// TIA Portal V16 program export: 1 tag tables, 0 data types, 0 data blocks, 2 code blocks (in call order from the OBs), 11 instance data blocks

VAR_GLOBAL   // PLC tag table "Standard-Variablentabelle"
   start AT %I0.4 : Bool;
   sensor1 AT %I0.0 : Bool;
   sensor2 AT %I0.1 : Bool;
   sensor3 AT %I0.2 : Bool;
   stop AT %I0.5 : Bool;
   "emergency stop" AT %I0.3 : Bool;
   "Detect Z" AT %I0.6 : Bool;
   movingx AT %I0.7 : Bool;
   movingz AT %I1.0 : Bool;
   rotating AT %I1.1 : Bool;
   "gripper rotating" AT %I1.2 : Bool;
   belt4m AT %Q0.0 : Bool;
   blet6m1 AT %Q0.1 : Bool;
   belt6m2 AT %Q0.2 : Bool;
   roller4m1 AT %Q0.3 : Bool;
   roller6m1 AT %Q0.4 : Bool;
   roller6m2 AT %Q0.5 : Bool;
   roller4m AT %Q0.6 : Bool;
   "Rob move x" AT %Q0.7 : Bool;
   "Rob move z" AT %Q1.0 : Bool;
   grab AT %Q1.1 : Bool;
   X AT %M0.0 : Bool;
   SBox AT %M0.1 : Bool;
   LBox AT %M0.2 : Bool;
   Pallet AT %M0.3 : Bool;
   Tag_3 AT %M7.0 : Bool;
   incrementer AT %MW1 : Int;
   Tag_1 AT %M7.1 : Bool;
   T1DN AT %M3.0 : Bool;
   T2DN AT %M3.1 : Bool;
   T3DN AT %M3.2 : Bool;
   T4DN AT %M3.3 : Bool;
   T5DN AT %M3.4 : Bool;
   T6DN AT %M3.5 : Bool;
   T7DN AT %M3.6 : Bool;
   T8DN AT %M3.7 : Bool;
   "Move Rollers" AT %M4.0 : Bool;
   Tag_2 AT %M7.2 : Bool;
   "Rob Start" AT %M7.3 : Bool;
   Tag_4 AT %M5.0 : Bool;
   Tag_5 AT %M5.1 : Bool;
   "Repeat cycle" AT %M4.1 : Bool;
   Tag_6 AT %M5.2 : Bool;
   "CYC DN" AT %M5.3 : Bool;
   "CTU1 DN" AT %M5.4 : Bool;
   Tag_7 AT %M5.5 : Bool;
   "Move rollers again" AT %M5.6 : Bool;
   Tag_8 AT %M5.7 : Bool;
   T_CTU1DN AT %M6.0 : Bool;
   "End Pallet" AT %M6.1 : Bool;
   Tag_9 AT %M6.2 : Bool;
   Tag_10 AT %M6.3 : Bool;
   "T0.1DN" AT %M6.4 : Bool;
   TCTDN AT %M6.5 : Bool;
END_VAR

ORGANIZATION_BLOCK "Main"   // OB1, LAD, ProgramCycle
TITLE = "Main Program Sweep (Cycle)"
{ S7_Optimized_Access := 'TRUE' }
AUTHOR : Islam_Abdulnasser
VERSION : 0.1
// stored: AutoNumber true, IsIECCheckEnabled false, SetENOAutomatically false
   VAR_INPUT
      Initial_Call : Bool;   // Initial call of this OB
      Remanence : Bool;   // =True, if remanent data are available
   END_VAR
   VAR_TEMP   // added for the SCL form of the ladder/FBD networks
      _w1 : Bool;
      _w2 : Bool;
      _w3 : Bool;
   END_VAR
BEGIN

REGION Network 1
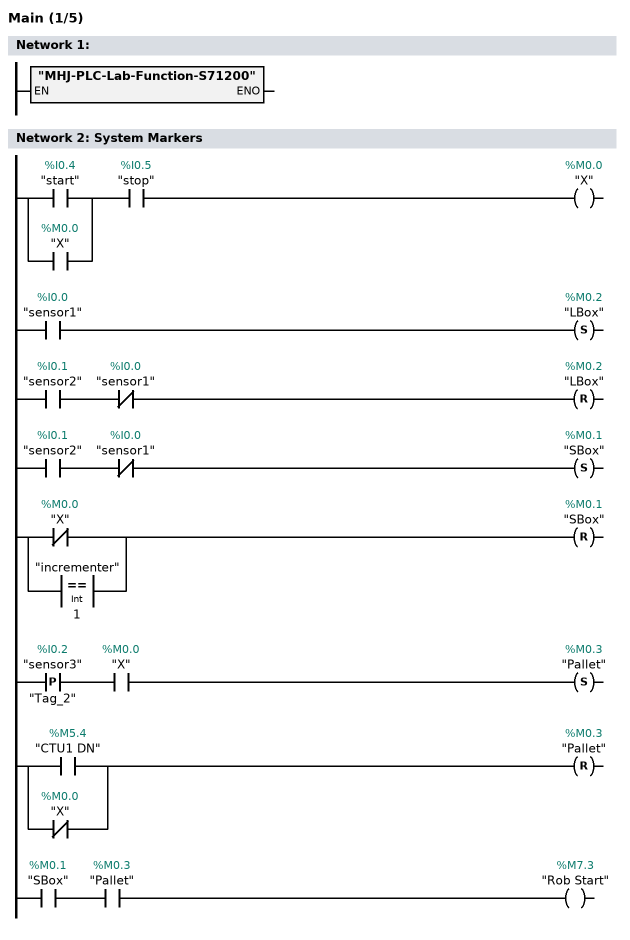
   RUNG wire#powerrail
      "MHJ-PLC-Lab-Function-S71200"()
   END_RUNG
   // the same network as SCL:
   "MHJ-PLC-Lab-Function-S71200"();
END_REGION

REGION Network 2: System Markers
   RUNG wire#powerrail
      Contact( "start" )
      wire#w1
      Contact( "stop" )
      Coil( "X" )
   END_RUNG
   RUNG wire#powerrail
      Contact( "X" )
   END_RUNG wire#w1
   RUNG wire#powerrail
      Contact( "sensor1" )
      S_Coil( "LBox" )
   END_RUNG
   RUNG wire#powerrail
      Contact( "sensor2" )
      I_Contact( "sensor1" )
      R_Coil( "LBox" )
   END_RUNG
   RUNG wire#powerrail
      Contact( "sensor2" )
      I_Contact( "sensor1" )
      S_Coil( "SBox" )
   END_RUNG
   RUNG wire#powerrail
      I_Contact( "X" )
      wire#w2
      R_Coil( "SBox" )
   END_RUNG
   RUNG wire#powerrail
      { S7_Templates := "SrcType := Int" } EQ_Contact(in1 := "incrementer", in2 := 1)
   END_RUNG wire#w2
   RUNG wire#powerrail
      P_Contact(operand := "sensor3", bit := "Tag_2")
      Contact( "X" )
      S_Coil( "Pallet" )
   END_RUNG
   RUNG wire#powerrail
      Contact( "CTU1 DN" )
      wire#w3
      R_Coil( "Pallet" )
   END_RUNG
   RUNG wire#powerrail
      I_Contact( "X" )
   END_RUNG wire#w3
   RUNG wire#powerrail
      Contact( "SBox" )
      Contact( "Pallet" )
      Coil( "Rob Start" )
   END_RUNG
   // the same network as SCL:
   "X" := ("start" OR "X") AND "stop";
   IF "sensor1" THEN "LBox" := TRUE; END_IF;
   IF "sensor2" AND NOT "sensor1" THEN
       "LBox" := FALSE;
       "SBox" := TRUE;
   END_IF;
   IF NOT "X" OR ("incrementer" = 1) THEN "SBox" := FALSE; END_IF;
   #_w1 := "sensor3" AND NOT "Tag_2";   // rising edge of "sensor3"
   "Tag_2" := "sensor3";
   IF #_w1 AND "X" THEN "Pallet" := TRUE; END_IF;
   IF "CTU1 DN" OR NOT "X" THEN "Pallet" := FALSE; END_IF;
   "Rob Start" := "SBox" AND "Pallet";
END_REGION

REGION Network 3: System Set
   // System Set
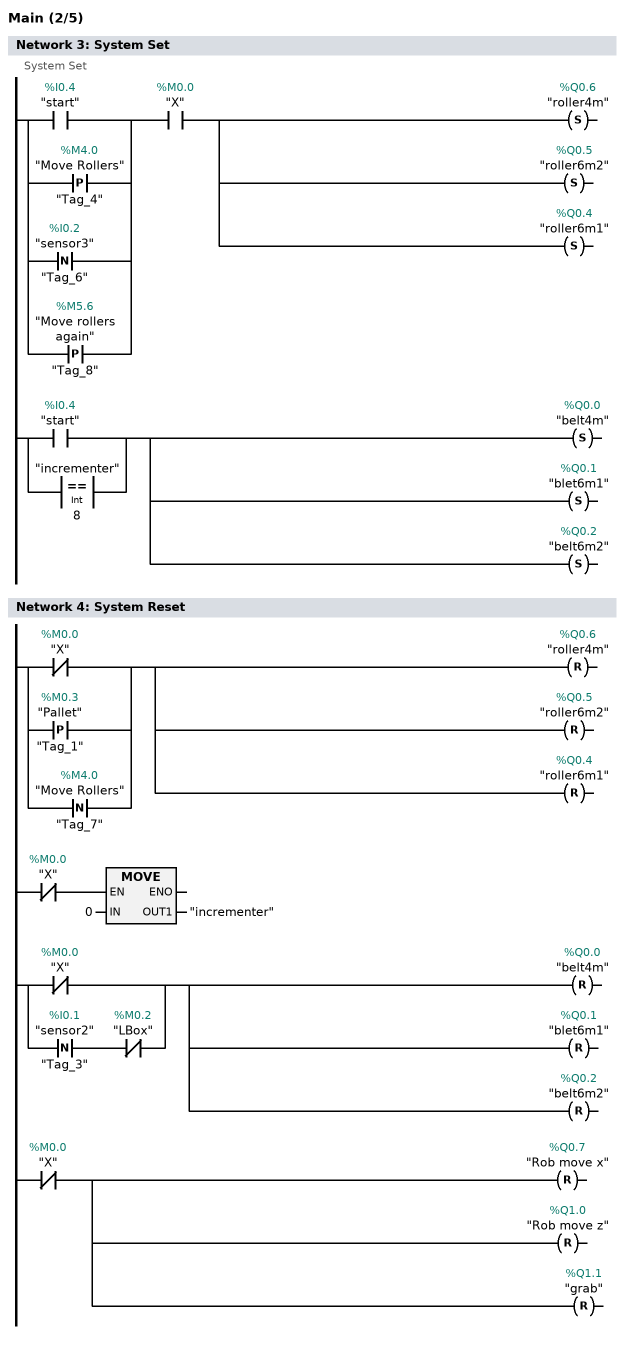
   RUNG wire#powerrail
      Contact( "start" )
      wire#w1
      Contact( "X" )
      wire#w2
      S_Coil( "roller4m" )
   END_RUNG
   RUNG wire#powerrail
      P_Contact(operand := "Move Rollers", bit := "Tag_4")
   END_RUNG wire#w1
   RUNG wire#powerrail
      N_Contact(operand := "sensor3", bit := "Tag_6")
   END_RUNG wire#w1
   RUNG wire#powerrail
      P_Contact(operand := "Move rollers again", bit := "Tag_8")
   END_RUNG wire#w1
   RUNG wire#w2
      S_Coil( "roller6m2" )
   END_RUNG
   RUNG wire#w2
      S_Coil( "roller6m1" )
   END_RUNG
   RUNG wire#powerrail
      Contact( "start" )
      wire#w3
      S_Coil( "belt4m" )
   END_RUNG
   RUNG wire#powerrail
      { S7_Templates := "SrcType := Int" } EQ_Contact(in1 := "incrementer", in2 := 8)
   END_RUNG wire#w3
   RUNG wire#w3
      S_Coil( "blet6m1" )
   END_RUNG
   RUNG wire#w3
      S_Coil( "belt6m2" )
   END_RUNG
   // the same network as SCL:
   #_w1 := "Move Rollers" AND NOT "Tag_4";   // rising edge of "Move Rollers"
   "Tag_4" := "Move Rollers";
   #_w2 := NOT "sensor3" AND "Tag_6";   // falling edge of "sensor3"
   "Tag_6" := "sensor3";
   #_w3 := "Move rollers again" AND NOT "Tag_8";   // rising edge of "Move rollers again"
   "Tag_8" := "Move rollers again";
   IF ("start" OR #_w1 OR #_w2 OR #_w3) AND "X" THEN
       "roller4m" := TRUE;
       "roller6m2" := TRUE;
       "roller6m1" := TRUE;
   END_IF;
   IF "start" OR ("incrementer" = 8) THEN
       "belt4m" := TRUE;
       "blet6m1" := TRUE;
       "belt6m2" := TRUE;
   END_IF;
END_REGION

REGION Network 4: System Reset
   RUNG wire#powerrail
      I_Contact( "X" )
      wire#w1
      R_Coil( "roller4m" )
   END_RUNG
   RUNG wire#powerrail
      P_Contact(operand := "Pallet", bit := "Tag_1")
   END_RUNG wire#w1
   RUNG wire#powerrail
      N_Contact(operand := "Move Rollers", bit := "Tag_7")
   END_RUNG wire#w1
   RUNG wire#w1
      R_Coil( "roller6m2" )
   END_RUNG
   RUNG wire#w1
      R_Coil( "roller6m1" )
   END_RUNG
   RUNG wire#powerrail
      I_Contact( "X" )
      Move(in := 0, out1 => "incrementer")
   END_RUNG
   RUNG wire#powerrail
      I_Contact( "X" )
      wire#w2
      R_Coil( "belt4m" )
   END_RUNG
   RUNG wire#powerrail
      N_Contact(operand := "sensor2", bit := "Tag_3")
      I_Contact( "LBox" )
   END_RUNG wire#w2
   RUNG wire#w2
      R_Coil( "blet6m1" )
   END_RUNG
   RUNG wire#w2
      R_Coil( "belt6m2" )
   END_RUNG
   RUNG wire#powerrail
      I_Contact( "X" )
      wire#w3
      R_Coil( "Rob move x" )
   END_RUNG
   RUNG wire#w3
      R_Coil( "Rob move z" )
   END_RUNG
   RUNG wire#w3
      R_Coil( "grab" )
   END_RUNG
   // the same network as SCL:
   #_w1 := "Pallet" AND NOT "Tag_1";   // rising edge of "Pallet"
   "Tag_1" := "Pallet";
   #_w2 := NOT "Move Rollers" AND "Tag_7";   // falling edge of "Move Rollers"
   "Tag_7" := "Move Rollers";
   IF NOT "X" OR #_w1 OR #_w2 THEN
       "roller4m" := FALSE;
       "roller6m2" := FALSE;
       "roller6m1" := FALSE;
   END_IF;
   IF NOT "X" THEN "incrementer" := 0; END_IF;
   #_w3 := NOT "sensor2" AND "Tag_3";   // falling edge of "sensor2"
   "Tag_3" := "sensor2";
   IF NOT "X" OR (#_w3 AND NOT "LBox") THEN
       "belt4m" := FALSE;
       "blet6m1" := FALSE;
       "belt6m2" := FALSE;
   END_IF;
   IF NOT "X" THEN
       "Rob move x" := FALSE;
       "Rob move z" := FALSE;
       "grab" := FALSE;
   END_IF;
END_REGION

REGION Network 5: Start Cycle
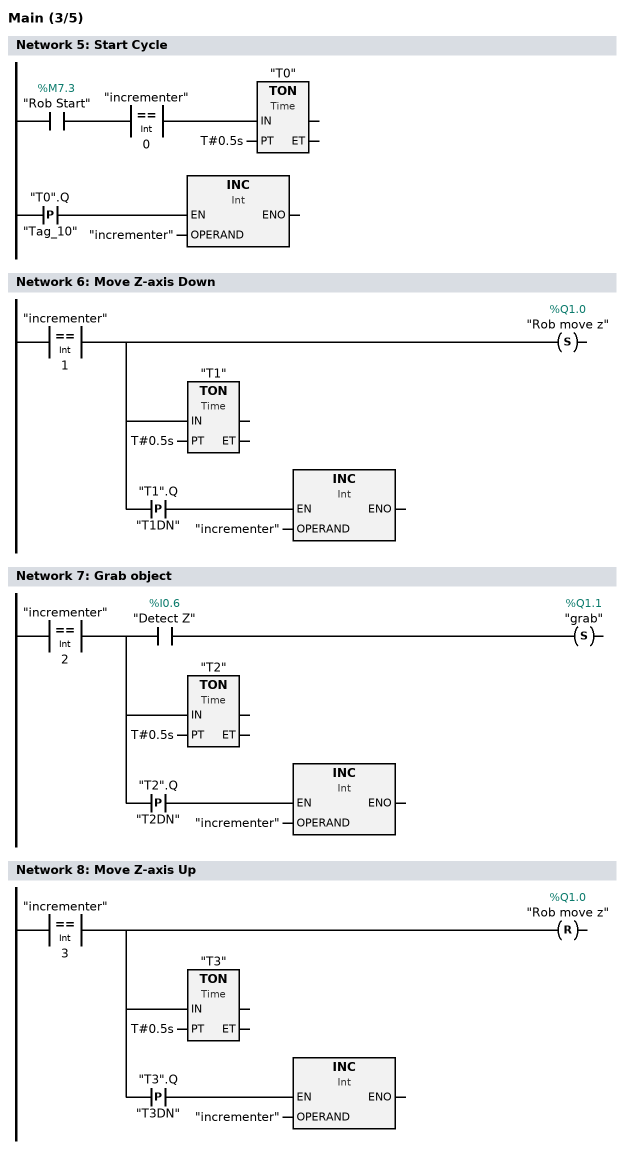
   RUNG wire#powerrail
      Contact( "Rob Start" )
      { S7_Templates := "SrcType := Int" } EQ_Contact(in1 := "incrementer", in2 := 0)
      { S7_Templates := "time_type := Time" } "T0".TON(pt := T#0.5s, et =>)
   END_RUNG
   RUNG wire#powerrail
      P_Contact(operand := "T0".Q, bit := "Tag_10")
      { S7_Templates := "DestType := Int" } Inc( "incrementer" )
   END_RUNG
   // the same network as SCL:
   "T0".TON(IN := "Rob Start" AND ("incrementer" = 0), PT := T#0.5s);
   #_w1 := "T0".Q AND NOT "Tag_10";   // rising edge of "T0".Q
   "Tag_10" := "T0".Q;
   IF #_w1 THEN "incrementer" := "incrementer" + 1; END_IF;
END_REGION

REGION Network 6: Move Z-axis Down
   RUNG wire#powerrail
      { S7_Templates := "SrcType := Int" } EQ_Contact(in1 := "incrementer", in2 := 1)
      wire#w1
      S_Coil( "Rob move z" )
   END_RUNG
   RUNG wire#w1
      { S7_Templates := "time_type := Time" } "T1".TON(pt := T#0.5s, et =>)
   END_RUNG
   RUNG wire#w1
      P_Contact(operand := "T1".Q, bit := "T1DN")
      { S7_Templates := "DestType := Int" } Inc( "incrementer" )
   END_RUNG
   // the same network as SCL:
   #_w1 := "incrementer" = 1;
   IF #_w1 THEN "Rob move z" := TRUE; END_IF;
   "T1".TON(IN := #_w1, PT := T#0.5s);
   #_w2 := #_w1 AND "T1".Q AND NOT "T1DN";   // rising edge of "T1".Q
   "T1DN" := "T1".Q;
   IF #_w2 THEN "incrementer" := "incrementer" + 1; END_IF;
END_REGION

REGION Network 7: Grab object
   RUNG wire#powerrail
      { S7_Templates := "SrcType := Int" } EQ_Contact(in1 := "incrementer", in2 := 2)
      wire#w1
      Contact( "Detect Z" )
      S_Coil( "grab" )
   END_RUNG
   RUNG wire#w1
      { S7_Templates := "time_type := Time" } "T2".TON(pt := T#0.5s, et =>)
   END_RUNG
   RUNG wire#w1
      P_Contact(operand := "T2".Q, bit := "T2DN")
      { S7_Templates := "DestType := Int" } Inc( "incrementer" )
   END_RUNG
   // the same network as SCL:
   #_w1 := "incrementer" = 2;
   IF #_w1 AND "Detect Z" THEN "grab" := TRUE; END_IF;
   "T2".TON(IN := #_w1, PT := T#0.5s);
   #_w2 := #_w1 AND "T2".Q AND NOT "T2DN";   // rising edge of "T2".Q
   "T2DN" := "T2".Q;
   IF #_w2 THEN "incrementer" := "incrementer" + 1; END_IF;
END_REGION

REGION Network 8: Move Z-axis Up
   RUNG wire#powerrail
      { S7_Templates := "SrcType := Int" } EQ_Contact(in1 := "incrementer", in2 := 3)
      wire#w1
      R_Coil( "Rob move z" )
   END_RUNG
   RUNG wire#w1
      { S7_Templates := "time_type := Time" } "T3".TON(pt := T#0.5s, et =>)
   END_RUNG
   RUNG wire#w1
      P_Contact(operand := "T3".Q, bit := "T3DN")
      { S7_Templates := "DestType := Int" } Inc( "incrementer" )
   END_RUNG
   // the same network as SCL:
   #_w1 := "incrementer" = 3;
   IF #_w1 THEN "Rob move z" := FALSE; END_IF;
   "T3".TON(IN := #_w1, PT := T#0.5s);
   #_w2 := #_w1 AND "T3".Q AND NOT "T3DN";   // rising edge of "T3".Q
   "T3DN" := "T3".Q;
   IF #_w2 THEN "incrementer" := "incrementer" + 1; END_IF;
END_REGION

REGION Network 9: Move X-axis Fowrard
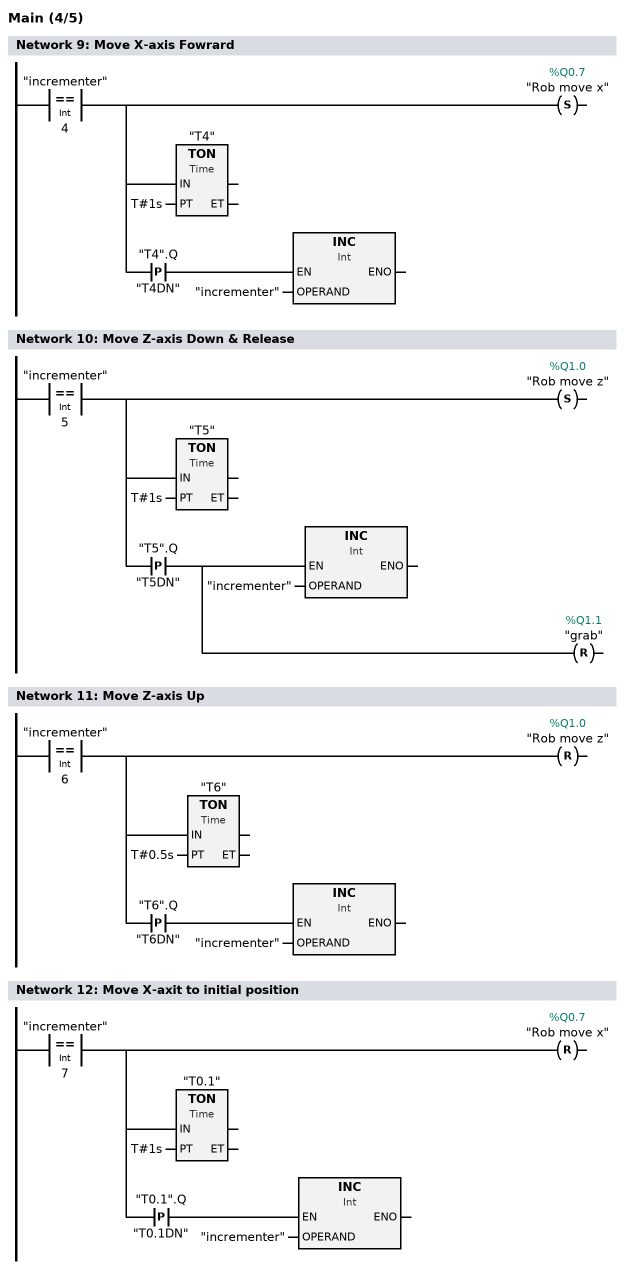
   RUNG wire#powerrail
      { S7_Templates := "SrcType := Int" } EQ_Contact(in1 := "incrementer", in2 := 4)
      wire#w1
      S_Coil( "Rob move x" )
   END_RUNG
   RUNG wire#w1
      { S7_Templates := "time_type := Time" } "T4".TON(pt := T#1s, et =>)
   END_RUNG
   RUNG wire#w1
      P_Contact(operand := "T4".Q, bit := "T4DN")
      { S7_Templates := "DestType := Int" } Inc( "incrementer" )
   END_RUNG
   // the same network as SCL:
   #_w1 := "incrementer" = 4;
   IF #_w1 THEN "Rob move x" := TRUE; END_IF;
   "T4".TON(IN := #_w1, PT := T#1s);
   #_w2 := #_w1 AND "T4".Q AND NOT "T4DN";   // rising edge of "T4".Q
   "T4DN" := "T4".Q;
   IF #_w2 THEN "incrementer" := "incrementer" + 1; END_IF;
END_REGION

REGION Network 10: Move Z-axis Down & Release
   RUNG wire#powerrail
      { S7_Templates := "SrcType := Int" } EQ_Contact(in1 := "incrementer", in2 := 5)
      wire#w1
      S_Coil( "Rob move z" )
   END_RUNG
   RUNG wire#w1
      { S7_Templates := "time_type := Time" } "T5".TON(pt := T#1s, et =>)
   END_RUNG
   RUNG wire#w1
      P_Contact(operand := "T5".Q, bit := "T5DN")
      wire#w2
      { S7_Templates := "DestType := Int" } Inc( "incrementer" )
   END_RUNG
   RUNG wire#w2
      R_Coil( "grab" )
   END_RUNG
   // the same network as SCL:
   #_w1 := "incrementer" = 5;
   IF #_w1 THEN "Rob move z" := TRUE; END_IF;
   "T5".TON(IN := #_w1, PT := T#1s);
   #_w2 := #_w1 AND "T5".Q AND NOT "T5DN";   // rising edge of "T5".Q
   "T5DN" := "T5".Q;
   IF #_w2 THEN
       "incrementer" := "incrementer" + 1;
       "grab" := FALSE;
   END_IF;
END_REGION

REGION Network 11: Move Z-axis Up
   RUNG wire#powerrail
      { S7_Templates := "SrcType := Int" } EQ_Contact(in1 := "incrementer", in2 := 6)
      wire#w1
      R_Coil( "Rob move z" )
   END_RUNG
   RUNG wire#w1
      { S7_Templates := "time_type := Time" } "T6".TON(pt := T#0.5s, et =>)
   END_RUNG
   RUNG wire#w1
      P_Contact(operand := "T6".Q, bit := "T6DN")
      { S7_Templates := "DestType := Int" } Inc( "incrementer" )
   END_RUNG
   // the same network as SCL:
   #_w1 := "incrementer" = 6;
   IF #_w1 THEN "Rob move z" := FALSE; END_IF;
   "T6".TON(IN := #_w1, PT := T#0.5s);
   #_w2 := #_w1 AND "T6".Q AND NOT "T6DN";   // rising edge of "T6".Q
   "T6DN" := "T6".Q;
   IF #_w2 THEN "incrementer" := "incrementer" + 1; END_IF;
END_REGION

REGION Network 12: Move X-axit to initial position
   RUNG wire#powerrail
      { S7_Templates := "SrcType := Int" } EQ_Contact(in1 := "incrementer", in2 := 7)
      wire#w1
      R_Coil( "Rob move x" )
   END_RUNG
   RUNG wire#w1
      { S7_Templates := "time_type := Time" } "T0.1".TON(pt := T#1s, et =>)
   END_RUNG
   RUNG wire#w1
      P_Contact(operand := "T0.1".Q, bit := "T0.1DN")
      { S7_Templates := "DestType := Int" } Inc( "incrementer" )
   END_RUNG
   // the same network as SCL:
   #_w1 := "incrementer" = 7;
   IF #_w1 THEN "Rob move x" := FALSE; END_IF;
   "T0.1".TON(IN := #_w1, PT := T#1s);
   #_w2 := #_w1 AND "T0.1".Q AND NOT "T0.1DN";   // rising edge of "T0.1".Q
   "T0.1DN" := "T0.1".Q;
   IF #_w2 THEN "incrementer" := "incrementer" + 1; END_IF;
END_REGION

REGION Network 13: Move Rollers a bit
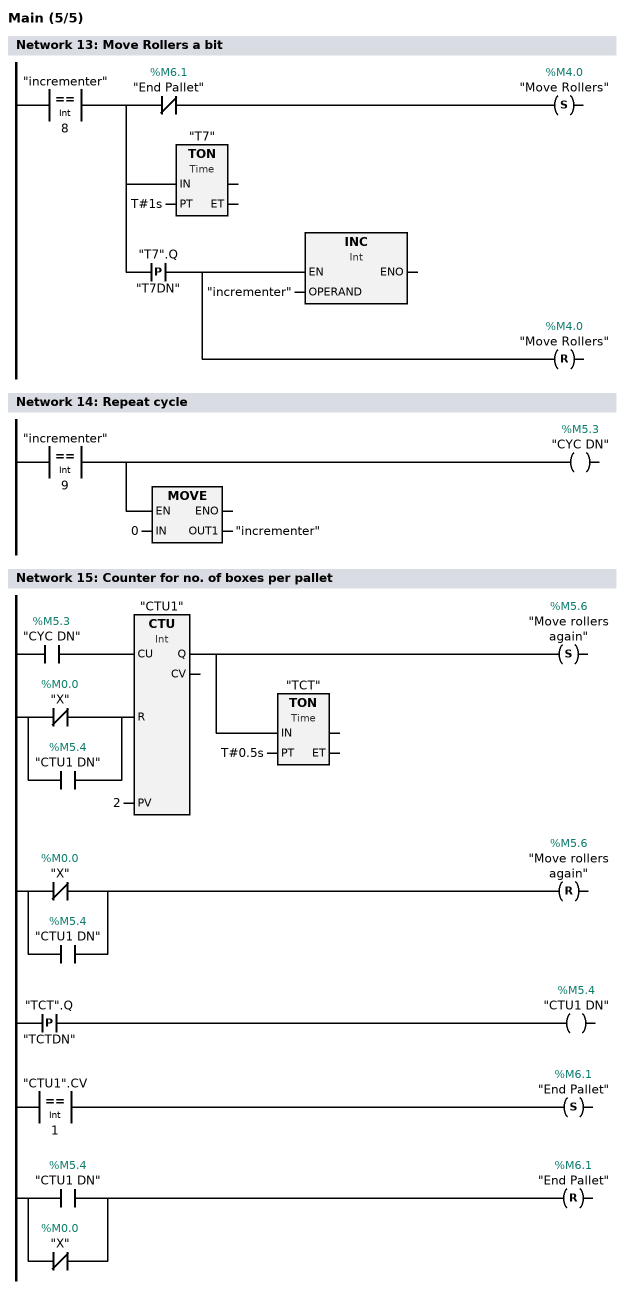
   RUNG wire#powerrail
      { S7_Templates := "SrcType := Int" } EQ_Contact(in1 := "incrementer", in2 := 8)
      wire#w1
      I_Contact( "End Pallet" )
      S_Coil( "Move Rollers" )
   END_RUNG
   RUNG wire#w1
      { S7_Templates := "time_type := Time" } "T7".TON(pt := T#1s, et =>)
   END_RUNG
   RUNG wire#w1
      P_Contact(operand := "T7".Q, bit := "T7DN")
      wire#w2
      { S7_Templates := "DestType := Int" } Inc( "incrementer" )
   END_RUNG
   RUNG wire#w2
      R_Coil( "Move Rollers" )
   END_RUNG
   // the same network as SCL:
   #_w1 := "incrementer" = 8;
   IF #_w1 AND NOT "End Pallet" THEN "Move Rollers" := TRUE; END_IF;
   "T7".TON(IN := #_w1, PT := T#1s);
   #_w2 := #_w1 AND "T7".Q AND NOT "T7DN";   // rising edge of "T7".Q
   "T7DN" := "T7".Q;
   IF #_w2 THEN
       "incrementer" := "incrementer" + 1;
       "Move Rollers" := FALSE;
   END_IF;
END_REGION

REGION Network 14: Repeat cycle
   RUNG wire#powerrail
      { S7_Templates := "SrcType := Int" } EQ_Contact(in1 := "incrementer", in2 := 9)
      wire#w1
      Coil( "CYC DN" )
   END_RUNG
   RUNG wire#w1
      Move(in := 0, out1 => "incrementer")
   END_RUNG
   // the same network as SCL:
   "CYC DN" := "incrementer" = 9;
   IF "CYC DN" THEN "incrementer" := 0; END_IF;
END_REGION

REGION Network 15: Counter for no. of boxes per pallet
   RUNG wire#powerrail
      Contact( "CYC DN" )
      { S7_Templates := "value_type := Int" } "CTU1".CTU(r := wire#w1, pv := 2, cv =>)
      wire#w2
      S_Coil( "Move rollers again" )
   END_RUNG
   RUNG wire#powerrail
      I_Contact( "X" )
   END_RUNG wire#w1
   RUNG wire#powerrail
      Contact( "CTU1 DN" )
   END_RUNG wire#w1
   RUNG wire#w2
      { S7_Templates := "time_type := Time" } "TCT".TON(pt := T#0.5s, et =>)
   END_RUNG
   RUNG wire#powerrail
      I_Contact( "X" )
      wire#w3
      R_Coil( "Move rollers again" )
   END_RUNG
   RUNG wire#powerrail
      Contact( "CTU1 DN" )
   END_RUNG wire#w3
   RUNG wire#powerrail
      P_Contact(operand := "TCT".Q, bit := "TCTDN")
      Coil( "CTU1 DN" )
   END_RUNG
   RUNG wire#powerrail
      { S7_Templates := "SrcType := Int" } EQ_Contact(in1 := "CTU1".CV, in2 := 1)
      S_Coil( "End Pallet" )
   END_RUNG
   RUNG wire#powerrail
      Contact( "CTU1 DN" )
      wire#w4
      R_Coil( "End Pallet" )
   END_RUNG
   RUNG wire#powerrail
      I_Contact( "X" )
   END_RUNG wire#w4
   // the same network as SCL:
   "CTU1".CTU(CU := "CYC DN", R := NOT "X" OR "CTU1 DN", PV := 2);
   IF "CTU1".Q THEN "Move rollers again" := TRUE; END_IF;
   "TCT".TON(IN := "CTU1".Q, PT := T#0.5s);
   IF NOT "X" OR "CTU1 DN" THEN "Move rollers again" := FALSE; END_IF;
   #_w1 := "TCT".Q AND NOT "TCTDN";   // rising edge of "TCT".Q
   "TCTDN" := "TCT".Q;
   "CTU1 DN" := #_w1;
   IF "CTU1".CV = 1 THEN "End Pallet" := TRUE; END_IF;
   IF "CTU1 DN" OR NOT "X" THEN "End Pallet" := FALSE; END_IF;
END_REGION
END_ORGANIZATION_BLOCK

FUNCTION "MHJ-PLC-Lab-Function-S71200" : Void
{ S7_Optimized_Access := 'TRUE' }
VERSION : 0.1
   VAR_TEMP 
      rdTimeReturn : Int;
      outputTime {InstructionName := 'DTL'; LibVersion := '1.0'} : DTL;
      SyncVal : Byte;
      forVal : Int;
      forVal_2 : Int;
      Value : Byte;
   END_VAR

   VAR CONSTANT 
      CompVal : Byte := 16#34;
      Value_01 : Byte := 16#11;
      Value_01_DW : DWord := 16#A165_D992;
      Value_02_DW : DWord := 16#58BE_4401;
   END_VAR


BEGIN
	
	#Value:=PEEK(area := 16#82,
	     dbNumber := 0,
	     byteOffset := 511);
	#Value := #Value + 1;
	
	POKE(area := 16#82,
	     dbNumber := 0,
	     byteOffset := 511,
	     value := #Value);
	
	POKE(area:=16#81,
	     dbNumber:=0,
	     byteOffset:=1016,
	     value:=#Value_01_DW);
	POKE(area := 16#81,
	     dbNumber := 0,
	     byteOffset := 1020,
	     value := #Value_02_DW);
	
	POKE(area := 16#81,
	     dbNumber := 0,
	     byteOffset := 511,
	     value := B#16#00);
	
	FOR #forVal := 0 TO 120 DO
	    FOR #forVal_2:=0 TO 10 DO
	        #rdTimeReturn:=RD_SYS_T(#outputTime);
	        #rdTimeReturn := WR_SYS_T(#outputTime);
	        #rdTimeReturn := RD_SYS_T(#outputTime);
	        #rdTimeReturn := WR_SYS_T(#outputTime);
	    END_FOR;
	    #SyncVal:= PEEK(area := 16#81,
	                   dbNumber := 0,
	                   byteOffset := 511);
	    IF #SyncVal = #CompVal THEN
	       GOTO M_1;
	    END_IF;
	END_FOR;
	RETURN;
	
	M_1:
	POKE(area := 16#81,
	     dbNumber := 0,
	     byteOffset := 511,
	     value := B#16#0);
	
	
	    
END_FUNCTION

DATA_BLOCK "CTU1"   // DB10
{ S7_Optimized_Access := 'TRUE' }
// stored: AutoNumber true, InstanceOfName IEC_COUNTER, OfSystemLibElement IEC_COUNTER, OfSystemLibVersion 1.0
"IEC_COUNTER"
   // VAR RETAIN
   //    CU : Bool;
   //    CD : Bool;
   //    R : Bool;
   //    LD : Bool;
   //    QU : Bool;
   //    QD : Bool;
   //    PV : Int;
   //    CV : Int;
   // END_VAR
BEGIN
END_DATA_BLOCK

DATA_BLOCK "T0.1"   // DB9
{ S7_Optimized_Access := 'TRUE' }
// stored: AutoNumber true, InstanceOfName IEC_TIMER, OfSystemLibElement IEC_TIMER, OfSystemLibVersion 1.0
"IEC_TIMER"
   // VAR
   //    PT : Time;
   //    ET { ExternalWritable := 'False'} : Time;
   //    IN : Bool;
   //    Q { ExternalWritable := 'False'} : Bool;
   // END_VAR
BEGIN
END_DATA_BLOCK

DATA_BLOCK "T0"   // DB8
{ S7_Optimized_Access := 'TRUE' }
// stored: AutoNumber true, InstanceOfName IEC_TIMER, OfSystemLibElement IEC_TIMER, OfSystemLibVersion 1.0
"IEC_TIMER"
   // VAR
   //    PT : Time;
   //    ET { ExternalWritable := 'False'} : Time;
   //    IN : Bool;
   //    Q { ExternalWritable := 'False'} : Bool;
   // END_VAR
BEGIN
END_DATA_BLOCK

DATA_BLOCK "T1"   // DB2
{ S7_Optimized_Access := 'TRUE' }
// stored: AutoNumber true, InstanceOfName IEC_TIMER, OfSystemLibElement IEC_TIMER, OfSystemLibVersion 1.0
"IEC_TIMER"
   // VAR
   //    PT : Time;
   //    ET { ExternalWritable := 'False'} : Time;
   //    IN : Bool;
   //    Q { ExternalWritable := 'False'} : Bool;
   // END_VAR
BEGIN
END_DATA_BLOCK

DATA_BLOCK "T2"   // DB3
{ S7_Optimized_Access := 'TRUE' }
// stored: AutoNumber true, InstanceOfName IEC_TIMER, OfSystemLibElement IEC_TIMER, OfSystemLibVersion 1.0
"IEC_TIMER"
   // VAR
   //    PT : Time;
   //    ET { ExternalWritable := 'False'} : Time;
   //    IN : Bool;
   //    Q { ExternalWritable := 'False'} : Bool;
   // END_VAR
BEGIN
END_DATA_BLOCK

DATA_BLOCK "T3"   // DB4
{ S7_Optimized_Access := 'TRUE' }
// stored: AutoNumber true, InstanceOfName IEC_TIMER, OfSystemLibElement IEC_TIMER, OfSystemLibVersion 1.0
"IEC_TIMER"
   // VAR
   //    PT : Time;
   //    ET { ExternalWritable := 'False'} : Time;
   //    IN : Bool;
   //    Q { ExternalWritable := 'False'} : Bool;
   // END_VAR
BEGIN
END_DATA_BLOCK

DATA_BLOCK "T4"   // DB5
{ S7_Optimized_Access := 'TRUE' }
// stored: AutoNumber true, InstanceOfName IEC_TIMER, OfSystemLibElement IEC_TIMER, OfSystemLibVersion 1.0
"IEC_TIMER"
   // VAR
   //    PT : Time;
   //    ET { ExternalWritable := 'False'} : Time;
   //    IN : Bool;
   //    Q { ExternalWritable := 'False'} : Bool;
   // END_VAR
BEGIN
END_DATA_BLOCK

DATA_BLOCK "T5"   // DB6
{ S7_Optimized_Access := 'TRUE' }
// stored: AutoNumber true, InstanceOfName IEC_TIMER, OfSystemLibElement IEC_TIMER, OfSystemLibVersion 1.0
"IEC_TIMER"
   // VAR
   //    PT : Time;
   //    ET { ExternalWritable := 'False'} : Time;
   //    IN : Bool;
   //    Q { ExternalWritable := 'False'} : Bool;
   // END_VAR
BEGIN
END_DATA_BLOCK

DATA_BLOCK "T6"   // DB1
{ S7_Optimized_Access := 'TRUE' }
// stored: AutoNumber true, InstanceOfName IEC_TIMER, OfSystemLibElement IEC_TIMER, OfSystemLibVersion 1.0
"IEC_TIMER"
   // VAR
   //    PT : Time;
   //    ET { ExternalWritable := 'False'} : Time;
   //    IN : Bool;
   //    Q { ExternalWritable := 'False'} : Bool;
   // END_VAR
BEGIN
END_DATA_BLOCK

DATA_BLOCK "T7"   // DB7
{ S7_Optimized_Access := 'TRUE' }
// stored: AutoNumber true, InstanceOfName IEC_TIMER, OfSystemLibElement IEC_TIMER, OfSystemLibVersion 1.0
"IEC_TIMER"
   // VAR
   //    PT : Time;
   //    ET { ExternalWritable := 'False'} : Time;
   //    IN : Bool;
   //    Q { ExternalWritable := 'False'} : Bool;
   // END_VAR
BEGIN
END_DATA_BLOCK

DATA_BLOCK "TCT"   // DB11
{ S7_Optimized_Access := 'TRUE' }
// stored: AutoNumber true, InstanceOfName IEC_TIMER, OfSystemLibElement IEC_TIMER, OfSystemLibVersion 1.0
"IEC_TIMER"
   // VAR
   //    PT : Time;
   //    ET { ExternalWritable := 'False'} : Time;
   //    IN : Bool;
   //    Q { ExternalWritable := 'False'} : Bool;
   // END_VAR
BEGIN
END_DATA_BLOCK
